// TwinCAT 3 PLC project PLC1
// ProgramVersion: 3.1.4024.0
// libraries:
//   Tc2_Standard, * (Beckhoff Automation GmbH)
//   Tc2_System, * (Beckhoff Automation GmbH)
//   Tc3_Module, * (Beckhoff Automation GmbH)
//   VisuSymbols,3.5.10.0,System
// project tree:
//   / GlobalTextList.TcGTLO, PlcTask.TcTTO, Visualization Manager.TcVMO (not stored)
//   GVLs/ GVL.TcGVL
//   POUs/ MAIN.TcPOU, POU.TcPOU (not stored)
//   VISUs/ Visualization.TcVIS
// real-time tasks:
//   TASK PlcTask: cycle T#10ms, priority 6, ADS port 350

CONFIGURATION PLC1
    RESOURCE PLC ON TwinCAT3
        TASK PlcTask(INTERVAL := T#10ms, PRIORITY := 6);
        PROGRAM MAIN WITH PlcTask : MAIN;
    END_RESOURCE
END_CONFIGURATION

// ---- GVLs/GVL.TcGVL
{attribute 'qualified_only'}
VAR_GLOBAL
	mb_Input_Coils        : ARRAY [0..255] OF BOOL;
    mb_Output_Coils       : ARRAY [0..255] OF BOOL;
    mb_Input_Registers    : ARRAY [0..255] OF WORD;
    mb_Output_Registers   : ARRAY [0..255] OF WORD;
END_VAR

// ---- POUs/MAIN.TcPOU
PROGRAM MAIN
VAR
	resetButton : BOOL;
	buttonPressed : BOOL;
	LAMP : BOOL; //Box is present in the pick up area
	craneMoving : BOOL;
	craneControllerStarted : BOOL;
	craneIdle : BOOL;
	beltMoving : BOOL;
	beltStopped : BOOL;
END_VAR

IF (buttonPressed = TRUE) THEN  // Start the belt which kicks off everything
	GVL.mb_Input_Registers[0] := 1;
	beltMoving := TRUE;
END_IF
//Box detection logic, box detected send the signal to the crane to start moving
IF (GVL.mb_Output_Registers[0] = 1) THEN // Box detected
	GVL.mb_Input_Registers[1] := 1; //Box detected, write to webots to start crane controller
	beltStopped := TRUE;
	beltMoving := FALSE;
	LAMP := TRUE; // Box waiting for pickup
	craneControllerStarted := TRUE;
END_IF
//Box detection logic, box is not present
IF (GVL.mb_Output_Registers[0] = 0) THEN // No box detected
	GVL.mb_Input_Registers[1] := 0; // No box idle crane
	IF (GVL.mb_Input_Registers[0] = 1) THEN
	beltMoving := TRUE;
	beltStopped := FALSE;
	END_IF
	LAMP := FALSE; // No box waiting
END_IF
//Checking if the crane is moving
IF (GVL.mb_Output_Registers[1] = 1) THEN
	craneMoving := TRUE;
	IF (craneControllerStarted = TRUE) THEN
	craneIdle := FALSE;
	END_IF
END_IF
//Checking if the crane is idle
IF (GVL.mb_Output_Registers[1] = 0) THEN
	craneMoving := FALSE;
	IF (craneControllerStarted = TRUE) THEN
	craneIdle := TRUE;
	END_IF
END_IF
//Reset button
IF (resetButton = TRUE) THEN
	GVL.mb_Input_Registers[0] := 0;
	GVL.mb_Input_Registers[1] := 0;
	GVL.mb_Output_Registers[0] := 0;
	GVL.mb_Output_Registers[1] := 0;
	LAMP := FALSE;
	craneMoving := FALSE;
	craneControllerStarted := FALSE;
	craneIdle := FALSE;
	beltMoving := FALSE;
	beltStopped := FALSE;
END_IF

END_PROGRAM

// ---- GlobalTextList.TcGTLO
TEXTLIST GlobalTextList
  427 = 'Belt moving'
  248 = 'Belt stopped'
  509 = 'Box detected'
  23 = 'Crane controller started'
  558 = 'Crane idle'
  667 = 'Crane in motion'
  235 = 'Reset'
  858 = 'Start'
  750 = 'Start Belt'
END_TEXTLIST

// ---- VISUs/Visualization.TcVIS
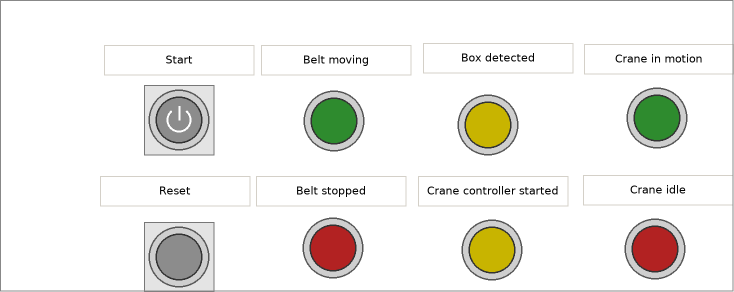
VISUALIZATION Visualization  // 734x292
    Lamp1 (453,90 70x70), variable: MAIN.LAMP, style: Lamp-Lamp1-Yellow
    PowerSwitch (144,85 70x70), variable: MAIN.buttonPressed, behaviour: TOGGLE, style: Switch-PowerSwitch-Gray
    Textfield (104,45 150x30), "Start"
    Textfield (423,43 150x30), "Box detected"
    Lamp1 (457,215 70x70), variable: MAIN.craneControllerStarted, style: Lamp-Lamp1-Yellow
    Textfield (418,176 150x30), "Crane controller started"
    Lamp1 (622,83 70x70), variable: MAIN.craneMoving, style: Lamp-Lamp1-Green
    Textfield (584,44 150x30), "Crane in motion"
    PushSwitch (144,222 70x70), variable: MAIN.resetButton, behaviour: TOGGLE, style: Switch-PushSwitch-Gray
    Textfield (100,176 150x30), "Reset"
    Lamp1 (620,214 70x70), variable: MAIN.craneIdle, style: Lamp-Lamp1-Red
    Textfield (583,175 150x30), "Crane idle"
    Lamp1 (299,86 70x70), variable: MAIN.beltMoving, style: Lamp-Lamp1-Green
    Lamp1 (298,213 70x70), variable: MAIN.beltStopped, style: Lamp-Lamp1-Red
    Textfield (261,45 150x30), "Belt moving"
    Textfield (256,176 150x30), "Belt stopped"
END_VISUALIZATION
